PROGRAM main
VAR
	Sensor_Input AT %IX0.0 : bool;
	Reset_Switch AT %IX0.1 : bool;
	Full_Box_Alarm AT %QX0.0 : bool;
	CTU0 : CTU;
END_VAR

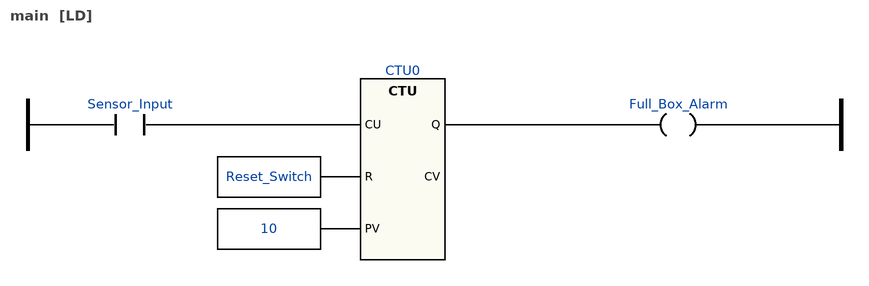
(* LD diagram, written out as Structured Text *)
CTU0(CU := Sensor_Input, R := Reset_Switch, PV := 10);
Full_Box_Alarm := CTU0.Q;
END_PROGRAM
